Fanuc KAREL source: V_LED_ON.kl

PROGRAM T
%NOLOCKGROUP
VAR
 v0 : INTEGER
 v1 : INTEGER
 v2 : INTEGER
BEGIN
 V_LED_ON(v0, v1, v2)
END T
